// TIA Portal V19 export
VAR_GLOBAL   // PLC tag table "D12"
   D12_Lp_EntryReq_LB202 AT %Q108.4 : Bool;   // 231SH1
   D12_Lp_SafetyReset_LB202 AT %Q108.5 : Bool;   // 231SH2
   D12_Pb_EntryReq_LB202 AT %I107.0 : Bool;   // 231SH1
   D12_Pb_SafetyReset_LB202 AT %I107.1 : Bool;   // 231SH2
   D12_Comando_Elettroserratura AT %Q108.3 : Bool;   // 23102
   D12_Cancello_Chiuso AT %I106.6 : Bool;   // 23101
   D12_Cancello_Bloccato AT %I106.7 : Bool;   // 23103
   D12_Ls_Os1 AT %I1072.2 : Bool;   // 105DI2 - 231A1
   D12_Ls_Os2 AT %I1072.6 : Bool;   // 105DI6 - 231A1
END_VAR
